(* IEC 61131-3 sources: inj-machine-docs/docs, 3 files *)

(* ---- 中子定义.st ---- *)
TYPE E_CoreState :
(
    (* 状态机枚举 *)
	eState_Idle,				// 空闲状态
	eState_Init,				// 初始化
	eState_CoreIning,			// 中子进中
	eState_CoreIned,			// 中子进完成
	eState_CoreOuting,			// 中子退中
	eState_CoreOuted,			// 中子退完成
	eState_Error				// 错误状态

);
END_TYPE

TYPE ST_CoreSeg :
STRUCT

	(* 单段工艺参数 *)
	uiPres: UINT;			// 设定压力
	uiSpd: UINT;			// 设定速度
	uiTime: UINT;			// 设定停止时间
	uiCount: UINT;			// 设定停止计数

END_STRUCT
END_TYPE

TYPE ST_CorePara :
STRUCT

	(* 中子进工艺参数 14*)
	uiCoreInStartMode: UINT;		// 中子进开始方式 0:行程 1:位置
	uiCoreInStroke: UINT;			// 中子进开始行程
	udiCoreInPos: UDINT;			// 中子进开始位置
	uiCoreInStopMode: UINT;			// 中子进停止方式 0:时间 1:行程 2:计数
	uiCoreInLimitTime: UINT;		// 中子进限制时间
	stCoreInSeg: ST_CoreSeg;		// 中子进设定参数

	uiCoreInPresStartGrad: UINT;			// 压力启动斜率
	uiCoreInPresStopGrad: UINT;				// 压力停止斜率
	uiCoreInSpdStartGrad: UINT;				// 速度启动斜率
	uiCoreInSpdStopGrad: UINT;				// 速度停止斜率

	(* 中子退工艺参数 14*)
	uiCoreOutStartMode: UINT;		// 中子退开始方式 0:行程 1:位置
	uiCoreOutStroke: UINT;			// 中子退开始行程
	udiCoreOutPos: UDINT;			// 中子退开始位置
	uiCoreOutStopMode: UINT;		// 中子退停止方式 0:时间 1:行程 2:计数
	uiCoreOutLimitTime: UINT;		// 中子退限制时间
	stCoreOutSeg: ST_CoreSeg;		// 中子退设定参数

	uiCoreOutPresStartGrad: UINT;			// 压力启动斜率
	uiCoreOutPresStopGrad: UINT;			// 压力停止斜率
	uiCoreOutSpdStartGrad: UINT;			// 速度启动斜率
	uiCoreOutSpdStopGrad: UINT;				// 速度停止斜率

END_STRUCT
END_TYPE

FUNCTION_BLOCK FB_Core
VAR_IN_OUT
	stCoreAxis: ST_AxisRefHyd;
END_VAR
VAR_INPUT

    (* 控制命令 *)
	bStart: BOOL;				// 启动
	bStop: BOOL;				// 停止(有减速停)
	bEStop: BOOL;				// 急停(立即停止，无减速停)
	bReset: BOOL;				// 复位

    (* 模式选择 *)
	uiCoreMode: UINT;		// 0:无模式 1:中子进模式 2:中子退模式

	(* 上位机设定参数输入 *)
	stCorePara: ST_CorePara;

	(* 数字信号输入 *)
	bCoreInStop: BOOL;			// 中子进停止
	bCoreOutStop: BOOL;			// 中子退停止

	(* 模拟信号输入 *)

END_VAR
VAR_OUTPUT

	(* 状态输出 *)
	bBusy: BOOL;		// 忙状态
	bDone: BOOL;		// 完成状态
	bAlarm: BOOL;		// 报警状态

    (* 报警信息 *)
	uiAlarmID: UINT;		// 报警代码
							(*	0:无
								1000:
								1001:中子进未定时完成
								1002:中子退未定时完成
							*)

    (* 动作提示 *)
	uiActHint: UINT;		// 当前动作状态
							(*	0:无动作	1:报警状态	  2:中子进完成  3:中子退完成
								10: 		11:中子进1段  12:			13:
								20:			21:中子退1段  22:  			23:
							*)
	uiActTime: UINT;		// 当前动作运行时间

	(* 动作状态输出 *)
	bCoreIned: BOOL;		// 中子进完成
	bCoreOuted: BOOL;		// 中子退完成

    (* 控制命令输出 *)
	uiPresCmd: UINT;		// 压力命令输出
	uiSpdCmd: UINT;			// 速度命令输出
	udiPosCmd: UDINT;		// 位置命令输出

END_VAR

(* ---- 储料定义.st ---- *)
TYPE E_MeterState :
(
    (* 状态机枚举 *)
	eState_Idle,				// 空闲状态
	eState_Init,				// 初始化
	eState_Metering,			// 储料中(8段)
	eState_Metered,				// 储料完成
	eState_Error				// 错误状态

);
END_TYPE

TYPE ST_MeterSeg :
STRUCT

	(* 单段工艺参数 *)
	uiSPres: UINT;		// 设定压力
	uiBackPres: UINT;	// 设定背压
	uiSpd: UINT;		// 设定速度
	udiPos: UDINT;		// 设定位置
	uiPresGrad: UINT;	// 设定压力斜率
	uiSpdGrad: UINT;	// 设定速度斜率

END_STRUCT
END_TYPE

TYPE ST_MeterPara :
STRUCT

	(* 储料工艺参数 71*)
	uiMeterSegCnt: UINT;						// 储料段数选择
	uiMeterMode: UINT;							// 储料退方式选择 0:电子尺  1:行程
	uiMeterLimitTime: UINT;						// 储料限制时间
	aMeterSeg: ARRAY[1..8] OF ST_MeterSeg;		// 储料多段设定参数

	uiMeterPresStartGrad: UINT;			// 压力启动斜率
	uiMeterPresStopGrad: UINT;			// 压力停止斜率
	uiMeterSpdStartGrad: UINT;			// 速度启动斜率
	uiMeterSpdStopGrad: UINT;			// 速度停止斜率

END_STRUCT
END_TYPE

FUNCTION_BLOCK FB_Meter
VAR_IN_OUT
	stMeterAxis: ST_AxisRefHyd;
END_VAR
VAR_INPUT

    (* 控制命令 *)
	bStart: BOOL;				// 启动
	bStop: BOOL;				// 停止(有减速停)
	bEStop: BOOL;				// 急停(立即停止，无减速停)
	bReset: BOOL;				// 复位

    (* 模式选择 *)
// 	uiMeterMode: UINT;		// 0:无模式 1: 2: 3:

	(* 上位机设定参数输入 *)
	stMeterPara: ST_MeterPara;

	(* 数字信号输入 *)
	bMeterStop: BOOL;			// 储料停止

	(* 模拟信号输入 *)
	udiInjElecRulerVal: UDINT;			// 射胶电子尺值

END_VAR
VAR_OUTPUT

	(* 状态输出 *)
	bBusy: BOOL;		// 忙状态
	bDone: BOOL;		// 完成状态
	bAlarm: BOOL;		// 报警状态

    (* 报警信息 *)
	uiAlarmID: UINT;		// 报警代码
							(*	0:无
								1000:
								1001:
								1002:
							*)

    (* 动作提示 *)
	uiActHint: UINT;		// 当前动作状态
							(*	0:无动作  1:报警状态  2:储料完成    3:
								10: 	  11:储料1段  12:储料2段	13: 储料3段  14:储料4段    15:储料5段  16: 储料6段  17:储料7段   18:储料8段
							*)
	uiActTime: UINT;		// 当前动作运行时间

	(* 动作状态输出 *)
	bMetered: BOOL;				//储料完成

    (* 控制命令输出 *)
	uiPresCmd: UINT;		// 压力命令输出
	uiBackPresCmd: UINT;	// 背压命令输出
	uiSpdCmd: UINT;			// 速度命令输出
	udiPosCmd: UDINT;		// 位置命令输出

END_VAR

(* ---- 射胶定义.st ---- *)
TYPE E_InjectState :
(
    (* 状态机枚举 *)
	eState_Idle,				// 空闲状态
	eState_Init,				// 初始化
	eState_Injecting,			// 射出中(10段)
	eState_Injected,			// 射出完成
	eState_Holding,				// 保压中(8段)
	eState_Held,				// 保压完成
	eState_SuckBacking,			// 射退中
	eState_SuckBacked,			// 射退完成
	eState_Error				// 错误状态
);
END_TYPE

TYPE ST_InjectSeg :
STRUCT

	(* 单段工艺参数 *)
	uiPres: UINT;		// 设定压力
	uiSpd: UINT;		// 设定速度
	udiPos: UDINT;		// 设定位置
	uiTime: UINT;		// 设定时间
	uiPresGrad: UINT;	// 设定压力斜率
	uiSpdGrad: UINT;	// 设定速度斜率

END_STRUCT
END_TYPE

TYPE ST_HoldSeg :
STRUCT

	(* 单段工艺参数 *)
	uiPres: UINT;		// 设定压力
	uiSpd: UINT;		// 设定速度
	uiTime: UINT;		// 设定时间

END_STRUCT
END_TYPE

TYPE ST_InjectPara :
STRUCT

	(* 射出多段工艺参数 79*)
	uiInjSegCnt: UINT;						// 射出段数选择
	uiInjMode: UINT;						// 射出方式选择 0:电子尺  1:行程  2:时间
	uiInjTotalTime: UINT;					// 射出总时间
	uiInjToHoldMode: UINT;					// 转保压方式
 	uiInjToHoldPres: UINT;					// 转保压压力
	aInjSeg: ARRAY[1..10] OF ST_InjectSeg;	// 射出多段设定参数

	uiInjPresStartGrad: UINT;				// 压力启动斜率
	uiInjPresStopGrad: UINT;				// 压力停止斜率
	uiInjSpdStartGrad: UINT;				// 速度启动斜率
	uiInjSpdStopGrad: UINT;					// 速度停止斜率

	(* 保压多段工艺参数 25*)
	uiHoldSegCnt: UINT;							// 保压段数选择
	aHoldSeg: ARRAY[1..8] OF ST_HoldSeg;		// 保压多段设定参数

	(* 射退工艺参数 12*)
	uiSuckBackMode: UINT;						// 射退方式选择 0:电子尺  1:时间(时间为0,走行程开关)
	stSuckBackSeg: ST_InjectSeg;				// 射退设定参数

	uiSuckBackPresStartGrad: UINT;				// 压力启动斜率
	uiSuckBackPresStopGrad: UINT;				// 压力停止斜率
	uiSuckBackSpdStartGrad: UINT;				// 速度启动斜率
	uiSuckBackSpdStopGrad: UINT;				// 速度停止斜率

END_STRUCT
END_TYPE

FUNCTION_BLOCK FB_Inject
VAR_IN_OUT
	stInjectAxis: ST_AxisRefHyd;
END_VAR
VAR_INPUT

    (* 控制命令 *)
	bStart: BOOL;				// 启动
	bStop: BOOL;				// 停止(有减速停)
	bEStop: BOOL;				// 急停(立即停止，无减速停)
	bReset: BOOL;				// 复位

    (* 模式选择 *)
	uiInjectMode: UINT;		// 0:无模式 1:射出模式 2:射退模式

	(* 上位机设定参数输入 *)
	stInjectPara: ST_InjectPara;

	(* 数字信号输入 *)
	bInjSeg1Stop: BOOL;			// 二级射出     射出1段结束
	bInjSeg2Stop: BOOL;			// 三级射出     射出2段结束
	bInjStop: BOOL;				// 射出停止
	bSuckBackStop: BOOL;		// 射退停止

	(* 模拟信号输入 *)
	udiInjElecRulerVal: UDINT;			// 射胶电子尺值

END_VAR
VAR_OUTPUT

	(* 状态输出 *)
	bBusy: BOOL;		// 忙状态
	bDone: BOOL;		// 完成状态
	bAlarm: BOOL;		// 报警状态

    (* 报警信息 *)
	uiAlarmID: UINT;		// 报警代码
							(*	0:无
								1000:
								1001:
								1002:
							*)

    (* 动作提示 *)
	uiActHint: UINT;		// 当前动作状态
							(*	0:无动作	1:报警状态	2:射出完成  3:保压完成	4:射退完成 5:射退中   6:		 7:射出10段
								10: 		11:射出1段  12:射出2段	13:射出3段  14:射出4段 15:射出5段 16:射出6段 17:射出7段 18:射出8段 19:射出9段
								20:			21:保压1段  22:保压2段  23:保压3段  24:保压4段 25:保压5段 26:保压6段 27:保压7段 28:保压8段
							*)
	uiActTime: UINT;		// 当前动作运行时间

	(* 动作状态输出 *)
	bInjected: BOOL;		// 射出完成
	bHeld: BOOL;			// 保压完成
	bSuckBacked: BOOL;		// 射退完成

    (* 控制命令输出 *)
	uiPresCmd: UINT;		// 压力命令输出
	uiSpdCmd: UINT;			// 速度命令输出
	udiPosCmd: UDINT;		// 位置命令输出

END_VAR
